// TIA Portal V18 export
// export: Created 2026-01-09T11:32:00.4628567Z, ExportSetting WithDefaults, DisplayName Totally Integrated Automation Portal, DisplayVersion V18 Update 5, DisplayName TIA Portal Openness, DisplayVersion V18 Update 5, DisplayName TIA Portal Teamcenter Gateway, DisplayVersion V18, DisplayName TIA Portal Version Control Interface, DisplayVersion V18, DisplayName SINAMICS Startdrive Advanced, DisplayVersion V18 SP2 Update 1, DisplayName SINAMICS Startdrive G110M, G120, G120C, G120D, G120P, G115D, DisplayVersion V18 SP2 Update 1, DisplayName SINAMICS Startdrive G130, G150, S120, S150, SINAMICS MV, S210, G220, S200, DisplayVersion V18 SP2 Update 1, DisplayName STEP 7 Professional, DisplayVersion V18 Update 5, DisplayName STEP 7 Safety, DisplayVersion V18, DisplayName WinCC Professional, DisplayVersion V18 Update 5
TagTable "V90"
  InterfaceV90_In_iInterlock : Bool  (%DB[V90DBNum].DBX0.0, CPU S71500-2PN_TP700, 500 ms)
  InterfaceV90_In_iManJog+ : Bool  (%DB[V90DBNum].DBX0.1, CPU S71500-2PN_TP700, 500 ms)
  InterfaceV90_In_iManJog- : Bool  (%DB[V90DBNum].DBX0.2, CPU S71500-2PN_TP700, 500 ms)
  InterfaceV90_In_iAutoStart : Bool  (%DB[V90DBNum].DBX0.3, CPU S71500-2PN_TP700, 500 ms)
  InterfaceV90_In_iHome : Bool  (%DB[V90DBNum].DBX0.4, CPU S71500-2PN_TP700, 500 ms)
  InterfaceV90_In_iCancelTask : Bool  (%DB[V90DBNum].DBX0.5, CPU S71500-2PN_TP700, 500 ms)
  InterfaceV90_In_iPauseTask : Bool  (%DB[V90DBNum].DBX0.6, CPU S71500-2PN_TP700, 500 ms)
  InterfaceV90_In_iManStart : Bool  (%DB[V90DBNum].DBX0.7, CPU S71500-2PN_TP700, 500 ms)
  InterfaceV90_In_iManListStart : Bool  (%DB[V90DBNum].DBX1.0, CPU S71500-2PN_TP700, 500 ms)
  InterfaceV90_In_iLimitSwitchActive : Bool  (%DB[V90DBNum].DBX1.1, CPU S71500-2PN_TP700, 500 ms)
  InterfaceV90_In_iLimitSoftActive : Bool  (%DB[V90DBNum].DBX1.2, CPU S71500-2PN_TP700, 500 ms)
  InterfaceV90_In_iRunningTimeout : Time  (%DB[V90DBNum].DBD2, CPU S71500-2PN_TP700, 500 ms)
  InterfaceV90_In_iHomingTimeout : Time  (%DB[V90DBNum].DBD6, CPU S71500-2PN_TP700, 500 ms)
  InterfaceV90_In_iAutoPosition : DInt  (%DB[V90DBNum].DBD10, CPU S71500-2PN_TP700, 100 ms)
  InterfaceV90_In_iAutoVelocity : Int  (%DB[V90DBNum].DBW14, CPU S71500-2PN_TP700, 500 ms)
  InterfaceV90_In_iManListPosition : DInt  (%DB[V90DBNum].DBD16, CPU S71500-2PN_TP700, 500 ms)
  InterfaceV90_In_iManListVelocity : Int  (%DB[V90DBNum].DBW20, CPU S71500-2PN_TP700, 500 ms)
  InterfaceV90_In_iManListNumber : Int  (%DB[V90DBNum].DBW22, CPU S71500-2PN_TP700, 500 ms)
  InterfaceV90_In_iManPosition : DInt  (%DB[V90DBNum].DBD24, CPU S71500-2PN_TP700, 500 ms)
  InterfaceV90_In_iManVelocity : Int  (%DB[V90DBNum].DBW28, CPU S71500-2PN_TP700, 500 ms)
  InterfaceV90_In_iMode : Int  (%DB[V90DBNum].DBW30, CPU S71500-2PN_TP700, 500 ms)
  InterfaceV90_Out_oReady : Bool  (%DB[V90DBNum].DBX32.0, CPU S71500-2PN_TP700, 500 ms)
  InterfaceV90_Out_oWarning : Bool  (%DB[V90DBNum].DBX32.1, CPU S71500-2PN_TP700, 500 ms)
  InterfaceV90_Out_oError : Bool  (%DB[V90DBNum].DBX32.2, CPU S71500-2PN_TP700, 500 ms)
  InterfaceV90_Out_oServoEnable : Bool  (%DB[V90DBNum].DBX32.4, CPU S71500-2PN_TP700, 500 ms)
  InterfaceV90_Out_oRunning : Bool  (%DB[V90DBNum].DBX32.5, CPU S71500-2PN_TP700, 500 ms)
  InterfaceV90_Out_oHoming : Bool  (%DB[V90DBNum].DBX32.6, CPU S71500-2PN_TP700, 500 ms)
  InterfaceV90_Out_oHomeRef : Bool  (%DB[V90DBNum].DBX32.7, CPU S71500-2PN_TP700, 500 ms)
  InterfaceV90_Out_oServoPosOK : Bool  (%DB[V90DBNum].DBX33.0, CPU S71500-2PN_TP700, 500 ms)
  InterfaceV90_Out_oErrorCode : Int  (%DB[V90DBNum].DBW34, CPU S71500-2PN_TP700, 500 ms)
  InterfaceV90_Out_oStatus : Int  (%DB[V90DBNum].DBW36, CPU S71500-2PN_TP700, 500 ms)
  InterfaceV90_Out_oActPosition : DInt  (%DB[V90DBNum].DBD38, CPU S71500-2PN_TP700, 100 ms)
  InterfaceV90_IO_ioManEnale : Bool  (%DB[V90DBNum].DBX46.0, CPU S71500-2PN_TP700, 500 ms)
  V90DBNum : Int  (1 s)
  InterfaceV90_Manual_Index : Int  (%DB[V90DBNum].DBW150, CPU S71500-2PN_TP700, 1 s)
  InterfaceV90_Out_oManualListPos : DInt  (%DB[V90DBNum].DBD42, CPU S71500-2PN_TP700, 1 s)
  InterfaceV90_Interlock_Case1 : Bool  (%DB[V90DBNum].DBX394.1, CPU S71500-2PN_TP700, 1 s)
  InterfaceV90_Interlock_Case2 : Bool  (%DB[V90DBNum].DBX394.2, CPU S71500-2PN_TP700, 1 s)
  InterfaceV90_Interlock_Case3 : Bool  (%DB[V90DBNum].DBX394.3, CPU S71500-2PN_TP700, 1 s)
  InterfaceV90_Interlock_Case4 : Bool  (%DB[V90DBNum].DBX394.4, CPU S71500-2PN_TP700, 1 s)
  InterfaceV90_Interlock_Case5 : Bool  (%DB[V90DBNum].DBX394.5, CPU S71500-2PN_TP700, 1 s)
  InterfaceV90_Interlock_Case6 : Bool  (%DB[V90DBNum].DBX394.6, CPU S71500-2PN_TP700, 1 s)
  InterfaceV90_Interlock_Case7 : Bool  (%DB[V90DBNum].DBX394.7, CPU S71500-2PN_TP700, 1 s)
  InterfaceV90_Interlock_Case8 : Bool  (%DB[V90DBNum].DBX395.0, CPU S71500-2PN_TP700, 1 s)
  InterfaceV90_In_Home Pos Pls : Bool  (%DB[V90DBNum].DBX400.0, CPU S71500-2PN_TP700, 500 ms)
  InterfaceV90_OUT_Arrow indication : Int  (%DB[V90DBNum].DBW402, CPU S71500-2PN_TP700, 100 ms)
  InterfaceV90_OUT_Process prompt : Int  (%DB[V90DBNum].DBW404, CPU S71500-2PN_TP700, 100 ms)
  InterfaceV90_OUT_Button prompt : Int  (%DB[V90DBNum].DBW406, CPU S71500-2PN_TP700, 500 ms)
